SYSTEM TestDPFB
  (* Version 1.0, 2023-10-16, ADMIN *)
  APPLICATION TestDPApp
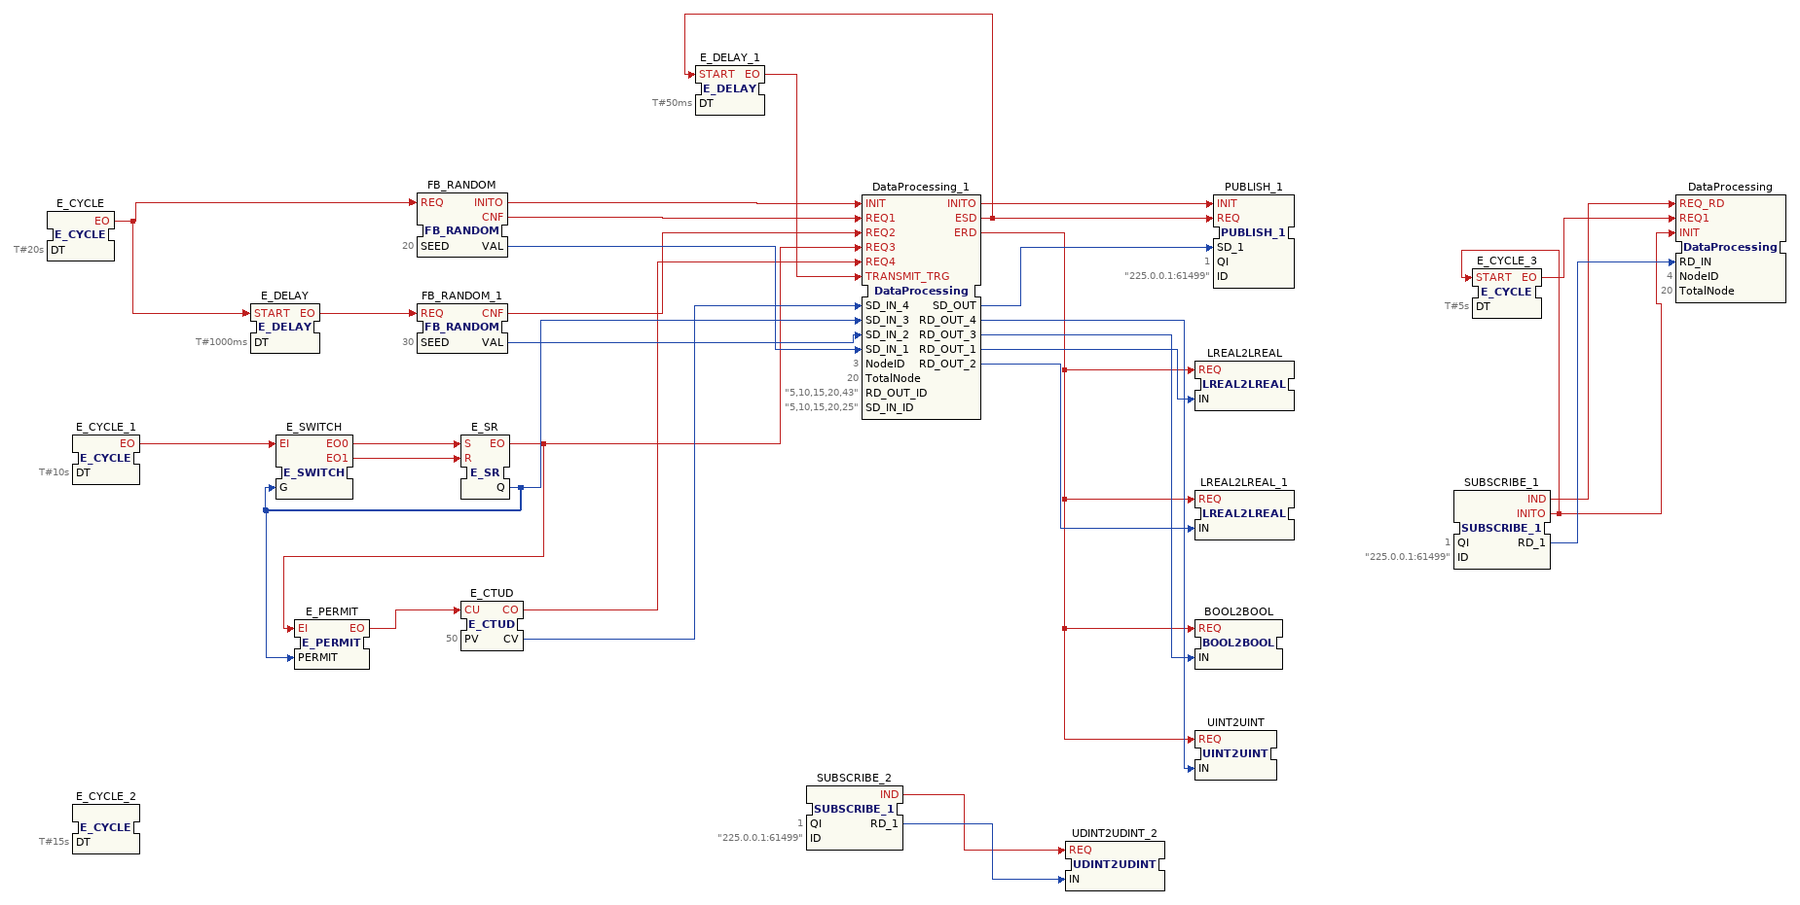
    FBS
      E_CYCLE : E_CYCLE(DT := T#20s);
      E_DELAY : E_DELAY(DT := T#1000ms);
      FB_RANDOM : FB_RANDOM(SEED := 20);
      FB_RANDOM_1 : FB_RANDOM(SEED := 30);
      E_SWITCH : E_SWITCH;
      E_SR : E_SR;
      E_CYCLE_1 : E_CYCLE(DT := T#10s);
      E_PERMIT : E_PERMIT;
      E_CTUD : E_CTUD(PV := 50);
      E_CYCLE_2 : E_CYCLE(DT := T#15s);
      SUBSCRIBE_1 : SUBSCRIBE_1(QI := 1, ID := "225.0.0.1:61499");
      PUBLISH_1 : PUBLISH_1(QI := 1, ID := "225.0.0.1:61499");
      DataProcessing_1 : DataProcessing(NodeID := 3, TotalNode := 20, RD_OUT_ID := "5,10,15,20,43", SD_IN_ID := "5,10,15,20,25");
      SUBSCRIBE_2 : SUBSCRIBE_1(QI := 1, ID := "225.0.0.1:61499");
      UDINT2UDINT_2 : UDINT2UDINT;
      DataProcessing : DataProcessing(NodeID := 4, TotalNode := 20);
      E_CYCLE_3 : E_CYCLE(DT := T#5s);
      E_DELAY_1 : E_DELAY(DT := T#50ms);
      UINT2UINT : UINT2UINT;
      BOOL2BOOL : BOOL2BOOL;
      LREAL2LREAL : LREAL2LREAL;
      LREAL2LREAL_1 : LREAL2LREAL;
    END_FBS
    EVENT_CONNECTIONS
      E_CYCLE.EO TO E_DELAY.START;
      E_CYCLE.EO TO FB_RANDOM.REQ;
      E_SWITCH.EO0 TO E_SR.S;
      E_SWITCH.EO1 TO E_SR.R;
      E_DELAY.EO TO FB_RANDOM_1.REQ;
      E_CYCLE_1.EO TO E_SWITCH.EI;
      E_SR.EO TO E_PERMIT.EI;
      E_PERMIT.EO TO E_CTUD.CU;
      DataProcessing_1.INITO TO PUBLISH_1.INIT;
      FB_RANDOM.INITO TO DataProcessing_1.INIT;
      FB_RANDOM.CNF TO DataProcessing_1.REQ1;
      FB_RANDOM_1.CNF TO DataProcessing_1.REQ2;
      E_SR.EO TO DataProcessing_1.REQ3;
      E_CTUD.CO TO DataProcessing_1.REQ4;
      SUBSCRIBE_2.IND TO UDINT2UDINT_2.REQ;
      SUBSCRIBE_1.IND TO DataProcessing.REQ_RD;
      DataProcessing_1.ESD TO PUBLISH_1.REQ;
      SUBSCRIBE_1.INITO TO E_CYCLE_3.START;
      E_CYCLE_3.EO TO DataProcessing.REQ1;
      SUBSCRIBE_1.INITO TO DataProcessing.INIT;
      DataProcessing_1.ESD TO E_DELAY_1.START;
      E_DELAY_1.EO TO DataProcessing_1.TRANSMIT_TRG;
      DataProcessing_1.ERD TO UINT2UINT.REQ;
      DataProcessing_1.ERD TO BOOL2BOOL.REQ;
      DataProcessing_1.ERD TO LREAL2LREAL.REQ;
      DataProcessing_1.ERD TO LREAL2LREAL_1.REQ;
    END_CONNECTIONS
    DATA_CONNECTIONS
      E_SR.Q TO E_SWITCH.G;
      E_SR.Q TO E_PERMIT.PERMIT;
      E_CTUD.CV TO DataProcessing_1.SD_IN_4;
      E_SR.Q TO DataProcessing_1.SD_IN_3;
      FB_RANDOM_1.VAL TO DataProcessing_1.SD_IN_2;
      FB_RANDOM.VAL TO DataProcessing_1.SD_IN_1;
      SUBSCRIBE_2.RD_1 TO UDINT2UDINT_2.IN;
      SUBSCRIBE_1.RD_1 TO DataProcessing.RD_IN;
      DataProcessing_1.SD_OUT TO PUBLISH_1.SD_1;
      DataProcessing_1.RD_OUT_4 TO UINT2UINT.IN;
      DataProcessing_1.RD_OUT_3 TO BOOL2BOOL.IN;
      DataProcessing_1.RD_OUT_1 TO LREAL2LREAL.IN;
      DataProcessing_1.RD_OUT_2 TO LREAL2LREAL_1.IN;
    END_CONNECTIONS
  END_APPLICATION
  DEVICE BeagleBoneBlack : BeagleBoneBlack(MGR_ID := "localhost:61499")
    {SET_ATTRIBUTE(Profile, HOLOBLOC)} (* device profile *)
    RESOURCE EMB_RES : EMB_RES
      FBS
        E_CYCLE : E_CYCLE(DT := T#20s);
        E_DELAY : E_DELAY(DT := T#1000ms);
        FB_RANDOM : FB_RANDOM(SEED := 20);
        FB_RANDOM_1 : FB_RANDOM(SEED := 30);
        E_SWITCH : E_SWITCH;
        E_SR : E_SR;
        E_CYCLE_1 : E_CYCLE(DT := T#10s);
        E_PERMIT : E_PERMIT;
        E_CTUD : E_CTUD(PV := 50);
        E_CYCLE_2 : E_CYCLE(DT := T#15s);
        PUBLISH_1 : PUBLISH_1(QI := 1, ID := "225.0.0.1:61499");
        DataProcessing_1 : DataProcessing(NodeID := 3, TotalNode := 20, RD_OUT_ID := "5,10,15,20,43", SD_IN_ID := "5,10,15,20,25");
        SUBSCRIBE_2 : SUBSCRIBE_1(QI := 1, ID := "225.0.0.1:61499");
        UDINT2UDINT_2 : UDINT2UDINT;
        E_DELAY_1 : E_DELAY(DT := T#50ms);
        UINT2UINT : UINT2UINT;
        BOOL2BOOL : BOOL2BOOL;
        LREAL2LREAL : LREAL2LREAL;
        LREAL2LREAL_1 : LREAL2LREAL;
      END_FBS
      EVENT_CONNECTIONS
        E_CYCLE.EO TO E_DELAY.START;
        E_CYCLE.EO TO FB_RANDOM.REQ;
        E_DELAY.EO TO FB_RANDOM_1.REQ;
        E_SWITCH.EO0 TO E_SR.S;
        E_SWITCH.EO1 TO E_SR.R;
        E_CYCLE_1.EO TO E_SWITCH.EI;
        START.COLD TO E_CYCLE.START;
        START.COLD TO FB_RANDOM.INIT;
        START.WARM TO E_CYCLE.START;
        START.WARM TO FB_RANDOM.INIT;
        START.COLD TO FB_RANDOM_1.INIT;
        START.WARM TO FB_RANDOM_1.INIT;
        START.COLD TO E_CYCLE_1.START;
        START.WARM TO E_CYCLE_1.START;
        E_SR.EO TO E_PERMIT.EI;
        E_PERMIT.EO TO E_CTUD.CU;
        START.COLD TO E_CYCLE_2.START;
        START.WARM TO E_CYCLE_2.START;
        DataProcessing_1.INITO TO PUBLISH_1.INIT;
        FB_RANDOM.INITO TO DataProcessing_1.INIT;
        FB_RANDOM.CNF TO DataProcessing_1.REQ1;
        FB_RANDOM_1.CNF TO DataProcessing_1.REQ2;
        E_SR.EO TO DataProcessing_1.REQ3;
        E_CTUD.CO TO DataProcessing_1.REQ4;
        SUBSCRIBE_2.IND TO UDINT2UDINT_2.REQ;
        DataProcessing_1.ESD TO PUBLISH_1.REQ;
        DataProcessing_1.ESD TO E_DELAY_1.START;
        E_DELAY_1.EO TO DataProcessing_1.TRANSMIT_TRG;
        DataProcessing_1.ERD TO UINT2UINT.REQ;
        DataProcessing_1.ERD TO BOOL2BOOL.REQ;
        DataProcessing_1.ERD TO LREAL2LREAL.REQ;
        DataProcessing_1.ERD TO LREAL2LREAL_1.REQ;
      END_CONNECTIONS
      DATA_CONNECTIONS
        E_SR.Q TO E_SWITCH.G;
        E_SR.Q TO E_PERMIT.PERMIT;
        E_CTUD.CV TO DataProcessing_1.SD_IN_4;
        E_SR.Q TO DataProcessing_1.SD_IN_3;
        FB_RANDOM_1.VAL TO DataProcessing_1.SD_IN_2;
        FB_RANDOM.VAL TO DataProcessing_1.SD_IN_1;
        SUBSCRIBE_2.RD_1 TO UDINT2UDINT_2.IN;
        DataProcessing_1.SD_OUT TO PUBLISH_1.SD_1;
        DataProcessing_1.RD_OUT_4 TO UINT2UINT.IN;
        DataProcessing_1.RD_OUT_3 TO BOOL2BOOL.IN;
        DataProcessing_1.RD_OUT_1 TO LREAL2LREAL.IN;
        DataProcessing_1.RD_OUT_2 TO LREAL2LREAL_1.IN;
      END_CONNECTIONS
    END_RESOURCE
  END_DEVICE
  DEVICE BeagleBoneBlack_1 : BeagleBoneBlack(MGR_ID := "localhost:61500")
    {SET_ATTRIBUTE(Profile, HOLOBLOC)} (* device profile *)
    RESOURCE EMB_RES : EMB_RES
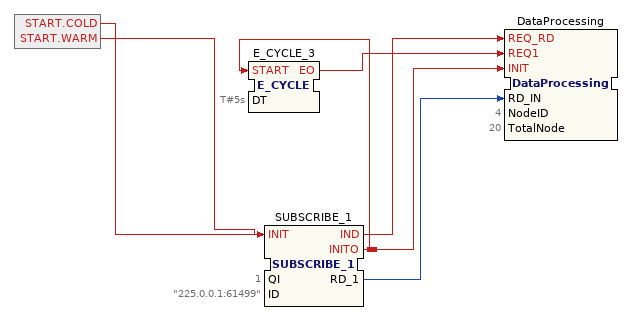
      FBS
        SUBSCRIBE_1 : SUBSCRIBE_1(QI := 1, ID := "225.0.0.1:61499");
        DataProcessing : DataProcessing(NodeID := 4, TotalNode := 20);
        E_CYCLE_3 : E_CYCLE(DT := T#5s);
      END_FBS
      EVENT_CONNECTIONS
        START.COLD TO SUBSCRIBE_1.INIT;
        START.WARM TO SUBSCRIBE_1.INIT;
        SUBSCRIBE_1.IND TO DataProcessing.REQ_RD;
        SUBSCRIBE_1.INITO TO E_CYCLE_3.START;
        E_CYCLE_3.EO TO DataProcessing.REQ1;
        SUBSCRIBE_1.INITO TO DataProcessing.INIT;
      END_CONNECTIONS
      DATA_CONNECTIONS
        SUBSCRIBE_1.RD_1 TO DataProcessing.RD_IN;
      END_CONNECTIONS
    END_RESOURCE
  END_DEVICE
  MAPPINGS
    TestDPApp.E_CYCLE ON BeagleBoneBlack.EMB_RES.E_CYCLE;
    TestDPApp.E_DELAY ON BeagleBoneBlack.EMB_RES.E_DELAY;
    TestDPApp.FB_RANDOM ON BeagleBoneBlack.EMB_RES.FB_RANDOM;
    TestDPApp.FB_RANDOM_1 ON BeagleBoneBlack.EMB_RES.FB_RANDOM_1;
    TestDPApp.E_SWITCH ON BeagleBoneBlack.EMB_RES.E_SWITCH;
    TestDPApp.E_SR ON BeagleBoneBlack.EMB_RES.E_SR;
    TestDPApp.E_CYCLE_1 ON BeagleBoneBlack.EMB_RES.E_CYCLE_1;
    TestDPApp.E_PERMIT ON BeagleBoneBlack.EMB_RES.E_PERMIT;
    TestDPApp.E_CTUD ON BeagleBoneBlack.EMB_RES.E_CTUD;
    TestDPApp.E_CYCLE_2 ON BeagleBoneBlack.EMB_RES.E_CYCLE_2;
    TestDPApp.PUBLISH_1 ON BeagleBoneBlack.EMB_RES.PUBLISH_1;
    TestDPApp.DataProcessing_1 ON BeagleBoneBlack.EMB_RES.DataProcessing_1;
    TestDPApp.SUBSCRIBE_1 ON BeagleBoneBlack_1.EMB_RES.SUBSCRIBE_1;
    TestDPApp.SUBSCRIBE_2 ON BeagleBoneBlack.EMB_RES.SUBSCRIBE_2;
    TestDPApp.UDINT2UDINT_2 ON BeagleBoneBlack.EMB_RES.UDINT2UDINT_2;
    TestDPApp.DataProcessing ON BeagleBoneBlack_1.EMB_RES.DataProcessing;
    TestDPApp.E_CYCLE_3 ON BeagleBoneBlack_1.EMB_RES.E_CYCLE_3;
    TestDPApp.E_DELAY_1 ON BeagleBoneBlack.EMB_RES.E_DELAY_1;
    TestDPApp.UINT2UINT ON BeagleBoneBlack.EMB_RES.UINT2UINT;
    TestDPApp.BOOL2BOOL ON BeagleBoneBlack.EMB_RES.BOOL2BOOL;
    TestDPApp.LREAL2LREAL ON BeagleBoneBlack.EMB_RES.LREAL2LREAL;
    TestDPApp.LREAL2LREAL_1 ON BeagleBoneBlack.EMB_RES.LREAL2LREAL_1;
  END_MAPPINGS
  SEGMENTS
    Ethernet : Ethernet;
  END_SEGMENTS
  LINKS
    BeagleBoneBlack => Ethernet;
    BeagleBoneBlack_1 => Ethernet;
  END_LINKS
END_SYSTEM
